// function block for inductive sensor with the option of debouncing + rising and falling edge detection.
FUNCTION_BLOCK FB_Component_InductiveSensor IMPLEMENTS  I_Component
VAR_INPUT
	bRawSignal		: BOOL;				// Raw input sensor
	tDebounce		: TIME := T#0MS;	// Debounce time
	tTimeout		: TIME := T#0MS;
	
	sName			: STRING[20];
	bEnable     	: BOOL;
END_VAR

VAR_OUTPUT
	bSensorActive	: BOOL;
	bTimeout		: BOOL;
	bRisingEdge		: BOOL;
	bFallingEdge	: BOOL;
	eState			: E_State;
	sStatusText 	: STRING[100];
END_VAR

VAR
	tDebounceTimer	: TON;
	tTimeoutTimer	: TON;
	
	bLastStableSignal	: BOOL := bRawSignal;
	bPendingSignal		: BOOL;
END_VAR

tDebounceTimer.PT 	:= tDebounce;
tTimeoutTimer.PT	:= tTimeout;

IF bEnable THEN
	CASE eState OF
		E_State.READY: 	IF bRawSignal <> bLastStableSignal THEN
										bPendingSignal := bRawSignal;
										eState := E_State.BUSY;
									ELSE
										tTimeoutTimer(IN := FALSE);
										tDebounceTimer(IN := FALSE);
									END_IF
									sStatusText := 'sensor active';
		
		E_State.BUSY:		tDebounceTimer(IN := TRUE);
									IF bRawSignal <> bPendingSignal THEN			// if signal bounces go back to ready state	
										eState := E_State.DONE;
									END_IF
			
									IF tDebounceTimer.Q THEN						// if signal stays stable for debounce duration -> trigger timeout
										eState := E_State.TIMEOUT;
									END_IF
									sStatusText := 'Debouncing sensor';
									
		E_State.TIMEOUT:	tTimeoutTimer(IN := TRUE);
									
									bRisingEdge  := NOT bLastStableSignal AND bPendingSignal;
	 								bFallingEdge := bLastStableSignal AND NOT bPendingSignal;
											
									bLastStableSignal := bPendingSignal;			// output stable signal
									bSensorActive	  := bLastStableSignal;
									IF tTimeoutTimer.Q THEN
										eState := E_State.DONE;
									END_IF
									sStatusText := 'sensor timeout';
			
		E_State.DONE:		tTimeoutTimer(IN := FALSE);
									tDebounceTimer(IN := FALSE);
	END_CASE
END_IF

METHOD M_Halt : BOOL
tDebounceTimer(IN := FALSE);
eState := E_State.HALTED;
END_METHOD

METHOD M_ResetEdge : BOOL
VAR_INPUT
END_VAR
bRisingEdge 	:= FALSE;
bFallingEdge	:= FALSE;
END_METHOD

METHOD M_Start : BOOL
IF eState <> E_State.BUSY AND eState <> E_State.TIMEOUT THEN
	eState := E_State.READY;
END_IF;
END_METHOD

METHOD M_Stop : BOOL
IF eState <> E_State.BUSY AND eState <> E_State.TIMEOUT  THEN
	eState := E_State.DONE;
END_IF
END_METHOD

END_FUNCTION_BLOCK

(* stored: Version 1.1.0.1, ProductVersion 3.1.4024.15
   POU FB_Component_InductiveSensor: Id {8e7ef9e5-be5c-4d5b-9caf-29f0d28584ab}, SpecialFunc None
   Method M_Halt: Id {f3238e3e-c657-463e-ba29-1e530a523711}
   Method M_ResetEdge: Id {c361819e-d8ca-4034-91ec-d2f2b326dd4e}
   Method M_Start: Id {332d80dd-0194-4918-b2f7-7e712950268d}
   Method M_Stop: Id {1e590e11-4492-46f6-8aed-701c371c3bb9} *)
